TYPE EL5152_ENC_ControlChannel :
STRUCT
	{attribute addProperty Name "Control"}
	Control AT %Q* : EL5152_Control;
	{attribute addProperty Name "Set counter value"}
	SetCounterValue AT %Q* : UINT;
END_STRUCT
END_TYPE

(* stored: Version 1.1.0.1, ProductVersion 3.1.4024.9
   DUT EL5152_ENC_ControlChannel: Id {b77e2c04-fc24-06bd-0572-7381fb17ef57} *)
